FUNCTION F_HelloWorld
VAR_INPUT
END_VAR
VAR
	nNum :DINT := 329;
END_VAR


		ADSLOGSTR(msgCtrlMask := ADSLOG_MSGTYPE_ERROR OR ADSLOG_MSGTYPE_LOG,
			msgFmtStr:= 'Hello world!!',
			strArg:='');
		ADSLOGDINT(msgCtrlMask := ADSLOG_MSGTYPE_WARN, msgFmtStr := 'value of num is %d', dintArg := nNum );

END_FUNCTION

(* stored: Version 1.1.0.1, ProductVersion 3.1.4024.16
   POU F_HelloWorld: Id {1b71dbe9-7d4c-445d-a8d7-fc2fe923832d}, SpecialFunc None *)
